(* IEC 61131-3 sources: RL_MAR/experiments/comparison/llm4plc/results/Qwen-Qwen3.5-9B_20260506_150728/20260506_165721, 4 files *)

(* ---- generated_code_iteration_0.st ---- *)
START_ST
FUNCTION_BLOCK CarParkingSystem
VAR_INPUT
    NewCarSlot : INT; (* Input for new car arrival slot number *)
END_VAR
VAR_OUTPUT
    Elevator1Busy : BOOL; (* Elevator 1 status - busy or idle *)
    Elevator2Busy : BOOL; (* Elevator 2 status - busy or idle *)
    Elevator1Position : INT; (* Elevator 1 current position *)
    Elevator2Position : INT; (* Elevator 2 current position *)
END_VAR
VAR
    (* FSM State Definitions *)
    CurrentState : INT; (* 0:IDLE_SCAN, 1:ASSIGN_TARGET, 2:MOVE_ELEVATOR_1, 3:MOVE_ELEVATOR_2, 4:COMPLETE_TASK *)

    (* Target and Status Variables *)
    Elevator1Target : INT; (* Elevator 1 target floor *)
    Elevator2Target : INT; (* Elevator 2 target floor *)
    SlotOccupied : BOOL; (* Temporary flag for the specific slot being processed *)
    TaskCompleted : BOOL; (* Temporary flag to indicate if movement is done *)

    (* Parking Slot Status Array *)
    CarSlots : ARRAY[1..100] OF BOOL; (* Array to represent parking slots - TRUE if occupied *)

    (* Simulation Variables for Movement *)
    MoveDirectionE1 : INT; (* Direction for Elevator 1: -1, 0, or 1 *)
    MoveDirectionE2 : INT; (* Direction for Elevator 2: -1, 0, or 1 *)
    MoveStepE1 : BOOL; (* Flag to simulate one step of movement for E1 *)
    MoveStepE2 : BOOL; (* Flag to simulate one step of movement for E2 *)
END_VAR
END_VAR

BEGIN
    (* --- INITIALIZATION --- *)
    IF CurrentState = 0 THEN
        (* Ensure initial state is clean on first execution or reset *)
        CurrentState := 0;
        Elevator1Target := 0;
        Elevator2Target := 0;
        MoveDirectionE1 := 0;
        MoveDirectionE2 := 0;
        MoveStepE1 := FALSE;
        MoveStepE2 := FALSE;
    END_IF;

    (* --- STATE 0: IDLE_SCAN --- *)
    (* System ready, no active tasks, waiting for NewCarSlot or checking for completed tasks *)
    IF CurrentState = 0 THEN
        Elevator1Busy := FALSE;
        Elevator2Busy := FALSE;

        (* Check if a new car has arrived *)
        IF NewCarSlot > 0 AND NewCarSlot <= 100 THEN
            (* Mark slot as occupied *)
            CarSlots[NewCarSlot] := TRUE;

            (* Determine which elevator to use based on slot range *)
            IF NewCarSlot <= 50 THEN
                (* Assign to Elevator 1 *)
                Elevator1Target := NewCarSlot;
                Elevator2Target := Elevator2Position; (* Keep E2 target as current position or 0 *)
                Elevator1Busy := TRUE;
                Elevator2Busy := FALSE;
                CurrentState := 2; (* Transition to MOVE_ELEVATOR_1 *)
            ELSE
                (* Assign to Elevator 2 *)
                Elevator1Target := Elevator1Position; (* Keep E1 target as current position or 0 *)
                Elevator2Target := NewCarSlot;
                Elevator1Busy := FALSE;
                Elevator2Busy := TRUE;
                CurrentState := 3; (* Transition to MOVE_ELEVATOR_2 *)
            END_IF;
        END_IF;

        (* Check if any task is completed and return to idle *)
        (* Note: In this FSM design, completion triggers a state change within the Move states,
           but we also check here to ensure state 0 is reached if logic dictates immediate reset *)
        IF Elevator1Busy = FALSE AND Elevator2Busy = FALSE THEN
            CurrentState := 0;
        END_IF;
    END_IF;

    (* --- STATE 1: ASSIGN_TARGET --- *)
    (* This state is logically merged into the transition logic above for efficiency.
       If NewCarSlot was processed, we moved to State 2 or 3.
       If no car arrived, we remain in State 0.
       We do not need a separate execution block for State 1 as the assignment happens instantly. *)

    (* --- STATE 2: MOVE_ELEVATOR_1 --- *)
    IF CurrentState = 2 THEN
        Elevator1Busy := TRUE;
        Elevator2Busy := FALSE;

        (* Simulate Movement Logic for Elevator 1 *)
        IF Elevator1Position < Elevator1Target THEN
            MoveDirectionE1 := 1;
        ELSIF Elevator1Position > Elevator1Target THEN
            MoveDirectionE1 := -1;
        ELSE
            MoveDirectionE1 := 0;
        END_IF;

        (* Simulate one step of movement *)
        IF MoveDirectionE1 <> 0 THEN
            Elevator1Position := Elevator1Position + MoveDirectionE1;
            (* Check if target reached *)
            IF Elevator1Position = Elevator1Target THEN
                TaskCompleted := TRUE;
                Elevator1Busy := FALSE;
                Elevator1Target := 0;
                CurrentState := 0; (* Transition to IDLE_SCAN *)
            END_IF;
        END_IF;
    END_IF;

    (* --- STATE 3: MOVE_ELEVATOR_2 --- *)
    IF CurrentState = 3 THEN
        Elevator1Busy := FALSE;
        Elevator2Busy := TRUE;

        (* Simulate Movement Logic for Elevator 2 *)
        IF Elevator2Position < Elevator2Target THEN
            MoveDirectionE2 := 1;
        ELSIF Elevator2Position > Elevator2Target THEN
            MoveDirectionE2 := -1;
        ELSE
            MoveDirectionE2 := 0;
        END_IF;

        (* Simulate one step of movement *)
        IF MoveDirectionE2 <> 0 THEN
            Elevator2Position := Elevator2Position + MoveDirectionE2;
            (* Check if target reached *)
            IF Elevator2Position = Elevator2Target THEN
                TaskCompleted := TRUE;
                Elevator2Busy := FALSE;
                Elevator2Target := 0;
                CurrentState := 0; (* Transition to IDLE_SCAN *)
            END_IF;
        END_IF;
    END_IF;

    (* --- STATE 4: COMPLETE_TASK --- *)
    (* This state is handled by the transition logic inside State 2 and State 3.
       Once the target is reached, the state is immediately reset to 0.
       No separate execution block is needed. *)

    (* --- END OF FUNCTION BLOCK --- *)
END_FUNCTION_BLOCK
END_ST

(* ---- generated_code_iteration_1.st ---- *)
START_REASON
The validation feedback indicates a CODESYS compiler error: "Unexpected token 'END_VAR'".
Analyzing the provided code:
1.  The code starts with `START_ST` and ends with `END_ST`.
2.  Inside the `FUNCTION_BLOCK CarParkingSystem`, there is a section defining variables:
    ```st
    VAR
        ...
    END_VAR
    END_VAR
    ```
    There are two `END_VAR` statements immediately following each other. The first one correctly closes the `VAR` section. The second one is extraneous and causes the syntax error.
3.  Additionally, the `FUNCTION_BLOCK` definition itself is missing the closing `END_FUNCTION_BLOCK` statement before the final `END_ST`. The code ends with `END_FUNCTION_BLOCK` inside the `END_ST` block, but looking closely at the provided text:
    ```st
    (* --- END OF FUNCTION BLOCK --- *)
    END_FUNCTION_BLOCK
    END_ST
    ```
    Wait, the provided code *does* have `END_FUNCTION_BLOCK`. Let me re-read the provided code block carefully.

    Provided code structure:
    ```st
    START_ST
    FUNCTION_BLOCK CarParkingSystem
    ...
    VAR
       ...
    END_VAR
    END_VAR  <-- ERROR 1: Duplicate END_VAR
    BEGIN
       ...
    END_FUNCTION_BLOCK
    END_ST
    ```

    Actually, looking at the very end of the user's input:
    ```st
    (* --- END OF FUNCTION BLOCK --- *)
    END_FUNCTION_BLOCK
    END_ST
    ```
    This looks correct structurally, except for the duplicate `END_VAR`.

    However, there is another potential issue. In IEC 61131-3, a `FUNCTION_BLOCK` must end with `END_FUNCTION_BLOCK`. The code has it.
    The specific error "Unexpected token 'END_VAR'" points directly to the line `END_VAR` appearing right after the first `END_VAR` that closes the `VAR` section.

    Correction Plan:
    1.  Remove the duplicate `END_VAR` after the variable declarations.
    2.  Ensure the `BEGIN` block is properly closed with `END_FUNCTION_BLOCK`.
    3.  Ensure the outer wrapper `START_ST` and `END_ST` are present.

    Let's double check the variable section in the input:
    ```st
    VAR
        (* FSM State Definitions *)
        CurrentState : INT; (* 0:IDLE_SCAN, 1:ASSIGN_TARGET, 2:MOVE_ELEVATOR_1, 3:MOVE_ELEVATOR_2, 4:COMPLETE_TASK *)

        (* Target and Status Variables *)
        Elevator1Target : INT; (* Elevator 1 target floor *)
        Elevator2Target : INT; (* Elevator 2 target floor *)
        SlotOccupied : BOOL; (* Temporary flag for the specific slot being processed *)
        TaskCompleted : BOOL; (* Temporary flag to indicate if movement is done *)

        (* Parking Slot Status Array *)
        CarSlots : ARRAY[1..100] OF BOOL; (* Array to represent parking slots - TRUE if occupied *)

        (* Simulation Variables for Movement *)
        MoveDirectionE1 : INT; (* Direction for Elevator 1: -1, 0, or 1 *)
        MoveDirectionE2 : INT; (* Direction for Elevator 2: -1, 0, or 1 *)
        MoveStepE1 : BOOL; (* Flag to simulate one step of movement for E1 *)
        MoveStepE2 : BOOL; (* Flag to simulate one step of movement for E2 *)
    END_VAR
    END_VAR  <-- This is the error.
    ```

    The fix is simply to delete the second `END_VAR`.

END_REASON

START_ST
FUNCTION_BLOCK CarParkingSystem
VAR_INPUT
    NewCarSlot : INT; (* Input for new car arrival slot number *)
END_VAR
VAR_OUTPUT
    Elevator1Busy : BOOL; (* Elevator 1 status - busy or idle *)
    Elevator2Busy : BOOL; (* Elevator 2 status - busy or idle *)
    Elevator1Position : INT; (* Elevator 1 current position *)
    Elevator2Position : INT; (* Elevator 2 current position *)
END_VAR
VAR
    (* FSM State Definitions *)
    CurrentState : INT; (* 0:IDLE_SCAN, 1:ASSIGN_TARGET, 2:MOVE_ELEVATOR_1, 3:MOVE_ELEVATOR_2, 4:COMPLETE_TASK *)

    (* Target and Status Variables *)
    Elevator1Target : INT; (* Elevator 1 target floor *)
    Elevator2Target : INT; (* Elevator 2 target floor *)
    SlotOccupied : BOOL; (* Temporary flag for the specific slot being processed *)
    TaskCompleted : BOOL; (* Temporary flag to indicate if movement is done *)

    (* Parking Slot Status Array *)
    CarSlots : ARRAY[1..100] OF BOOL; (* Array to represent parking slots - TRUE if occupied *)

    (* Simulation Variables for Movement *)
    MoveDirectionE1 : INT; (* Direction for Elevator 1: -1, 0, or 1 *)
    MoveDirectionE2 : INT; (* Direction for Elevator 2: -1, 0, or 1 *)
    MoveStepE1 : BOOL; (* Flag to simulate one step of movement for E1 *)
    MoveStepE2 : BOOL; (* Flag to simulate one step of movement for E2 *)
END_VAR
BEGIN
    (* --- INITIALIZATION --- *)
    IF CurrentState = 0 THEN
        (* Ensure initial state is clean on first execution or reset *)
        CurrentState := 0;
        Elevator1Target := 0;
        Elevator2Target := 0;
        MoveDirectionE1 := 0;
        MoveDirectionE2 := 0;
        MoveStepE1 := FALSE;
        MoveStepE2 := FALSE;
    END_IF;

    (* --- STATE 0: IDLE_SCAN --- *)
    (* System ready, no active tasks, waiting for NewCarSlot or checking for completed tasks *)
    IF CurrentState = 0 THEN
        Elevator1Busy := FALSE;
        Elevator2Busy := FALSE;

        (* Check if a new car has arrived *)
        IF NewCarSlot > 0 AND NewCarSlot <= 100 THEN
            (* Mark slot as occupied *)
            CarSlots[NewCarSlot] := TRUE;

            (* Determine which elevator to use based on slot range *)
            IF NewCarSlot <= 50 THEN
                (* Assign to Elevator 1 *)
                Elevator1Target := NewCarSlot;
                Elevator2Target := Elevator2Position; (* Keep E2 target as current position or 0 *)
                Elevator1Busy := TRUE;
                Elevator2Busy := FALSE;
                CurrentState := 2; (* Transition to MOVE_ELEVATOR_1 *)
            ELSE
                (* Assign to Elevator 2 *)
                Elevator1Target := Elevator1Position; (* Keep E1 target as current position or 0 *)
                Elevator2Target := NewCarSlot;
                Elevator1Busy := FALSE;
                Elevator2Busy := TRUE;
                CurrentState := 3; (* Transition to MOVE_ELEVATOR_2 *)
            END_IF;
        END_IF;

        (* Check if any task is completed and return to idle *)
        (* Note: In this FSM design, completion triggers a state change within the Move states,
           but we also check here to ensure state 0 is reached if logic dictates immediate reset *)
        IF Elevator1Busy = FALSE AND Elevator2Busy = FALSE THEN
            CurrentState := 0;
        END_IF;
    END_IF;

    (* --- STATE 1: ASSIGN_TARGET --- *)
    (* This state is logically merged into the transition logic above for efficiency.
       If NewCarSlot was processed, we moved to State 2 or 3.
       If no car arrived, we remain in State 0.
       We do not need a separate execution block for State 1 as the assignment happens instantly. *)

    (* --- STATE 2: MOVE_ELEVATOR_1 --- *)
    IF CurrentState = 2 THEN
        Elevator1Busy := TRUE;
        Elevator2Busy := FALSE;

        (* Simulate Movement Logic for Elevator 1 *)
        IF Elevator1Position < Elevator1Target THEN
            MoveDirectionE1 := 1;
        ELSIF Elevator1Position > Elevator1Target THEN
            MoveDirectionE1 := -1;
        ELSE
            MoveDirectionE1 := 0;
        END_IF;

        (* Simulate one step of movement *)
        IF MoveDirectionE1 <> 0 THEN
            Elevator1Position := Elevator1Position + MoveDirectionE1;
            (* Check if target reached *)
            IF Elevator1Position = Elevator1Target THEN
                TaskCompleted := TRUE;
                Elevator1Busy := FALSE;
                Elevator1Target := 0;
                CurrentState := 0; (* Transition to IDLE_SCAN *)
            END_IF;
        END_IF;
    END_IF;

    (* --- STATE 3: MOVE_ELEVATOR_2 --- *)
    IF CurrentState = 3 THEN
        Elevator1Busy := FALSE;
        Elevator2Busy := TRUE;

        (* Simulate Movement Logic for Elevator 2 *)
        IF Elevator2Position < Elevator2Target THEN
            MoveDirectionE2 := 1;
        ELSIF Elevator2Position > Elevator2Target THEN
            MoveDirectionE2 := -1;
        ELSE
            MoveDirectionE2 := 0;
        END_IF;

        (* Simulate one step of movement *)
        IF MoveDirectionE2 <> 0 THEN
            Elevator2Position := Elevator2Position + MoveDirectionE2;
            (* Check if target reached *)
            IF Elevator2Position = Elevator2Target THEN
                TaskCompleted := TRUE;
                Elevator2Busy := FALSE;
                Elevator2Target := 0;
                CurrentState := 0; (* Transition to IDLE_SCAN *)
            END_IF;
        END_IF;
    END_IF;

    (* --- STATE 4: COMPLETE_TASK --- *)
    (* This state is handled by the transition logic inside State 2 and State 3.
       Once the target is reached, the state is immediately reset to 0.
       No separate execution block is needed. *)

    (* --- END OF FUNCTION BLOCK --- *)
END_FUNCTION_BLOCK
END_ST

(* ---- generated_code_iteration_2.st ---- *)
START_REASON
The previous code failed the CODESYS compiler validation (Error 500: API call failed) despite passing ANTLR syntax checks. This usually indicates a logical structure error that a simple parser might miss but a compiler enforces strictly.

Analysis of the previous code:
1.  **Missing `VAR_INPUT`/`VAR_OUTPUT` Definitions in the `FUNCTION_BLOCK`**: The previous code block started with `FUNCTION_BLOCK CarParkingSystem` but immediately jumped into `VAR` (local variables) without defining `VAR_INPUT` or `VAR_OUTPUT`. In IEC 61131-3, a `FUNCTION_BLOCK` must explicitly define its interface (`VAR_INPUT`, `VAR_OUTPUT`, `VAR_IN_OUT`) before defining local variables (`VAR`).
2.  **Logic Flow Issue**: The previous code attempted to handle state transitions and output assignments within a single `BEGIN...END` block without a clear separation of interface definition and local logic. The compiler likely complained because it expected `VAR_INPUT` or `VAR_OUTPUT` after `FUNCTION_BLOCK` name but found `VAR` or `BEGIN` instead.
3.  **Redundant State Logic**: The previous logic tried to manage `Elevator1Busy` and `Elevator2Busy` inside the `BEGIN` block based on state, but since these are `VAR_OUTPUT`, they must be assigned at the end of the cycle or managed carefully. The previous code mixed state machine logic with output assignment in a way that might have caused a conflict or simply lacked the required interface section.

Correction Plan:
1.  Add `VAR_INPUT` and `VAR_OUTPUT` sections immediately after `FUNCTION_BLOCK CarParkingSystem`.
2.  Define the local variables (`VAR`) after the interface variables.
3.  Implement the Finite State Machine (FSM) logic cleanly.
4.  Ensure all outputs are assigned before the `END_FUNCTION_BLOCK`.
5.  Maintain the `START_ST` / `END_ST` wrapper.

END_REASON

START_ST
FUNCTION_BLOCK CarParkingSystem
VAR_INPUT
    NewCarSlot : INT;
END_VAR
VAR_OUTPUT
    Elevator1Busy : BOOL;
    Elevator2Busy : BOOL;
    Elevator1Position : INT;
    Elevator2Position : INT;
END_VAR
VAR
    (* FSM State Definitions *)
    CurrentState : INT; (* 0:IDLE_SCAN, 1:ASSIGN_TARGET, 2:MOVE_ELEVATOR_1, 3:MOVE_ELEVATOR_2, 4:COMPLETE_TASK *)

    (* Target and Status Variables *)
    Elevator1Target : INT;
    Elevator2Target : INT;
    SlotOccupied : BOOL;
    TaskCompleted : BOOL;

    (* Parking Slot Status Array *)
    CarSlots : ARRAY[1..100] OF BOOL;

    (* Simulation Variables for Movement *)
    MoveDirectionE1 : INT;
    MoveDirectionE2 : INT;
    MoveStepE1 : BOOL;
    MoveStepE2 : BOOL;
END_VAR

BEGIN
    (* --- INITIALIZATION --- *)
    IF CurrentState = 0 THEN
        CurrentState := 0;
        Elevator1Target := 0;
        Elevator2Target := 0;
        MoveDirectionE1 := 0;
        MoveDirectionE2 := 0;
        MoveStepE1 := FALSE;
        MoveStepE2 := FALSE;
    END_IF;

    (* --- STATE 0: IDLE_SCAN --- *)
    IF CurrentState = 0 THEN
        Elevator1Busy := FALSE;
        Elevator2Busy := FALSE;

        (* Check if a new car has arrived *)
        IF NewCarSlot > 0 AND NewCarSlot <= 100 THEN
            (* Mark slot as occupied *)
            CarSlots[NewCarSlot] := TRUE;

            (* Determine which elevator to use based on slot range *)
            IF NewCarSlot <= 50 THEN
                (* Assign to Elevator 1 *)
                Elevator1Target := NewCarSlot;
                Elevator2Target := Elevator2Position;
                CurrentState := 2; (* Transition to MOVE_ELEVATOR_1 *)
            ELSE
                (* Assign to Elevator 2 *)
                Elevator1Target := Elevator1Position;
                Elevator2Target := NewCarSlot;
                CurrentState := 3; (* Transition to MOVE_ELEVATOR_2 *)
            END_IF;
        END_IF;

        (* Check if any task is completed and return to idle *)
        IF Elevator1Busy = FALSE AND Elevator2Busy = FALSE THEN
            CurrentState := 0;
        END_IF;
    END_IF;

    (* --- STATE 2: MOVE_ELEVATOR_1 --- *)
    IF CurrentState = 2 THEN
        Elevator1Busy := TRUE;
        Elevator2Busy := FALSE;

        (* Simulate Movement Logic for Elevator 1 *)
        IF Elevator1Position < Elevator1Target THEN
            MoveDirectionE1 := 1;
        ELSIF Elevator1Position > Elevator1Target THEN
            MoveDirectionE1 := -1;
        ELSE
            MoveDirectionE1 := 0;
        END_IF;

        (* Simulate one step of movement *)
        IF MoveDirectionE1 <> 0 THEN
            Elevator1Position := Elevator1Position + MoveDirectionE1;
            (* Check if target reached *)
            IF Elevator1Position = Elevator1Target THEN
                TaskCompleted := TRUE;
                Elevator1Busy := FALSE;
                Elevator1Target := 0;
                CurrentState := 0; (* Transition to IDLE_SCAN *)
            END_IF;
        END_IF;
    END_IF;

    (* --- STATE 3: MOVE_ELEVATOR_2 --- *)
    IF CurrentState = 3 THEN
        Elevator1Busy := FALSE;
        Elevator2Busy := TRUE;

        (* Simulate Movement Logic for Elevator 2 *)
        IF Elevator2Position < Elevator2Target THEN
            MoveDirectionE2 := 1;
        ELSIF Elevator2Position > Elevator2Target THEN
            MoveDirectionE2 := -1;
        ELSE
            MoveDirectionE2 := 0;
        END_IF;

        (* Simulate one step of movement *)
        IF MoveDirectionE2 <> 0 THEN
            Elevator2Position := Elevator2Position + MoveDirectionE2;
            (* Check if target reached *)
            IF Elevator2Position = Elevator2Target THEN
                TaskCompleted := TRUE;
                Elevator2Busy := FALSE;
                Elevator2Target := 0;
                CurrentState := 0; (* Transition to IDLE_SCAN *)
            END_IF;
        END_IF;
    END_IF;

    (* --- STATE 1 & 4: HANDLED BY TRANSITIONS --- *)
    (* State 1 (Assign) and State 4 (Complete) are handled by the transitions
       within State 0, 2, and 3. No separate execution block needed. *)

END_FUNCTION_BLOCK
END_ST

(* ---- generated_code_iteration_3.st ---- *)
START_REASON
The previous code failed the CODESYS compiler validation with the specific error: "应该用';' 替换'IF'" (Should replace 'IF' with ';').

Analysis of the error:
1.  **Syntax Error in State Machine Logic**: The previous code structure used `IF CurrentState = 0 THEN ... END_IF;` followed by `IF CurrentState = 2 THEN ... END_IF;`. While this is valid ST syntax for sequential execution, the specific error message suggests a parsing issue often caused by missing semicolons at the end of statements or blocks within the `BEGIN...END` section, or a specific dialect requirement where the compiler expects a statement terminator before the next `IF` keyword in certain contexts (though standard IEC 61131-3 allows `IF` after `END_IF`).
2.  **Missing Semicolons**: A common cause for "replace IF with ;" errors in automated validation tools is that a preceding statement (like an assignment or a block) was missing its terminating semicolon `;` immediately before the next `IF` statement. For example, `END_IF` must be followed by `;` if it is not the last statement in the block, or the assignment inside the block might be missing a `;`.
3.  **Variable Initialization**: The variables `Elevator1Position` and `Elevator2Position` were used in the logic but not explicitly initialized in the `VAR` section or the initialization block, which can sometimes cause type inference errors in strict compilers if not handled carefully, though less likely to cause this specific syntax error.
4.  **Correction Strategy**:
    *   Ensure every single statement ends with a semicolon `;`.
    *   Explicitly initialize `Elevator1Position` and `Elevator2Position` to 0 in the `VAR` section or initialization logic to avoid undefined behavior.
    *   Simplify the state machine logic to ensure clear separation and proper termination of every block.
    *   Add the missing semicolons after `END_IF` statements that are not at the very end of the `BEGIN` block.

END_REASON

START_ST
FUNCTION_BLOCK CarParkingSystem
VAR_INPUT
    NewCarSlot : INT;
END_VAR
VAR_OUTPUT
    Elevator1Busy : BOOL;
    Elevator2Busy : BOOL;
    Elevator1Position : INT;
    Elevator2Position : INT;
END_VAR
VAR
    (* FSM State Definitions *)
    CurrentState : INT := 0; (* 0:IDLE_SCAN, 1:ASSIGN_TARGET, 2:MOVE_ELEVATOR_1, 3:MOVE_ELEVATOR_2, 4:COMPLETE_TASK *)

    (* Target and Status Variables *)
    Elevator1Target : INT;
    Elevator2Target : INT;
    SlotOccupied : BOOL;
    TaskCompleted : BOOL;

    (* Parking Slot Status Array *)
    CarSlots : ARRAY[1..100] OF BOOL;

    (* Simulation Variables for Movement *)
    MoveDirectionE1 : INT;
    MoveDirectionE2 : INT;
    MoveStepE1 : BOOL;
    MoveStepE2 : BOOL;

    (* Initial Positions *)
    InitPosE1 : INT := 0;
    InitPosE2 : INT := 0;
END_VAR

BEGIN
    (* --- INITIALIZATION --- *)
    IF CurrentState = 0 THEN
        CurrentState := 0;
        Elevator1Target := 0;
        Elevator2Target := 0;
        MoveDirectionE1 := 0;
        MoveDirectionE2 := 0;
        MoveStepE1 := FALSE;
        MoveStepE2 := FALSE;
        Elevator1Position := InitPosE1;
        Elevator2Position := InitPosE2;
    END_IF;

    (* --- STATE 0: IDLE_SCAN --- *)
    IF CurrentState = 0 THEN
        Elevator1Busy := FALSE;
        Elevator2Busy := FALSE;

        (* Check if a new car has arrived *)
        IF NewCarSlot > 0 AND NewCarSlot <= 100 THEN
            (* Mark slot as occupied *)
            CarSlots[NewCarSlot] := TRUE;

            (* Determine which elevator to use based on slot range *)
            IF NewCarSlot <= 50 THEN
                (* Assign to Elevator 1 *)
                Elevator1Target := NewCarSlot;
                Elevator2Target := Elevator2Position;
                CurrentState := 2; (* Transition to MOVE_ELEVATOR_1 *)
            ELSE
                (* Assign to Elevator 2 *)
                Elevator1Target := Elevator1Position;
                Elevator2Target := NewCarSlot;
                CurrentState := 3; (* Transition to MOVE_ELEVATOR_2 *)
            END_IF;
        END_IF;

        (* Check if any task is completed and return to idle *)
        IF Elevator1Busy = FALSE AND Elevator2Busy = FALSE THEN
            CurrentState := 0;
        END_IF;
    END_IF;

    (* --- STATE 2: MOVE_ELEVATOR_1 --- *)
    IF CurrentState = 2 THEN
        Elevator1Busy := TRUE;
        Elevator2Busy := FALSE;

        (* Simulate Movement Logic for Elevator 1 *)
        IF Elevator1Position < Elevator1Target THEN
            MoveDirectionE1 := 1;
        ELSIF Elevator1Position > Elevator1Target THEN
            MoveDirectionE1 := -1;
        ELSE
            MoveDirectionE1 := 0;
        END_IF;

        (* Simulate one step of movement *)
        IF MoveDirectionE1 <> 0 THEN
            Elevator1Position := Elevator1Position + MoveDirectionE1;
            (* Check if target reached *)
            IF Elevator1Position = Elevator1Target THEN
                TaskCompleted := TRUE;
                Elevator1Busy := FALSE;
                Elevator1Target := 0;
                CurrentState := 0; (* Transition to IDLE_SCAN *)
            END_IF;
        END_IF;
    END_IF;

    (* --- STATE 3: MOVE_ELEVATOR_2 --- *)
    IF CurrentState = 3 THEN
        Elevator1Busy := FALSE;
        Elevator2Busy := TRUE;

        (* Simulate Movement Logic for Elevator 2 *)
        IF Elevator2Position < Elevator2Target THEN
            MoveDirectionE2 := 1;
        ELSIF Elevator2Position > Elevator2Target THEN
            MoveDirectionE2 := -1;
        ELSE
            MoveDirectionE2 := 0;
        END_IF;

        (* Simulate one step of movement *)
        IF MoveDirectionE2 <> 0 THEN
            Elevator2Position := Elevator2Position + MoveDirectionE2;
            (* Check if target reached *)
            IF Elevator2Position = Elevator2Target THEN
                TaskCompleted := TRUE;
                Elevator2Busy := FALSE;
                Elevator2Target := 0;
                CurrentState := 0; (* Transition to IDLE_SCAN *)
            END_IF;
        END_IF;
    END_IF;

    (* --- STATE 1 & 4: HANDLED BY TRANSITIONS --- *)
    (* State 1 (Assign) and State 4 (Complete) are handled by the transitions
       within State 0, 2, and 3. No separate execution block needed. *)

END_FUNCTION_BLOCK
END_ST
